// Global constants
//
VAR_GLOBAL CONSTANT

	// Global constants...
	NUM_HISTORY_POINTS: INT := 120; // Amount of history points
	
END_VAR

(* stored: Version 1.1.0.1, ProductVersion 3.1.4022.6
   GVL Global_Constant: Id {a6cd0a2f-9c07-422f-97ea-67ac85e4b3bd} *)
